# EPICS autosave request: ipApp/Db/ADAM_4018p_settings.req
$(P)$(R):read.SCAN
$(P)$(R):readAll.SCAN
